TYPE ST_Params :
STRUCT
	fEncoderOffset : LREAL := 17574.8; 
	fGBtoDrumScaling : LREAL := 0.000744309; 
END_STRUCT
END_TYPE

(* stored: Version 1.1.0.1, ProductVersion 3.1.4024.12
   DUT ST_Params: Id {e00b6fa8-acf3-4801-a7dd-2cd3999ba2c8} *)
